Yaskawa INFORM job: FORLOOPTEST2.JBI

/JOB
//NAME FORLOOPTEST2
//POS
///NPOS 2,0,0,2,0,0
///TOOL 5
///POSTYPE PULSE
///PULSE
C00000=-3,-50477,-58433,3,-74931,486
C00001=-3,-50477,-58433,3,-74931,486
///POSTYPE ROBOT
///RECTAN
///RCONF 1,0,0,0,0,0,0,0,0,0,0,0,0,0,0,0,0,0,0,0,0,0,0,0
P00006=958.535,-37.777,-104.713,-165.2944,-7.1707,17.5149
P00007=956.377,3.321,-104.733,-165.2955,-7.1688,17.5107
//INST
///DATE 2024/03/06 15:14
///COMM For loop test
///ATTR SC,RW
///GROUP1 RB1
NOP
MOVJ C00000 VJ=3.00
FOR I001 START= 5 TO 7
	 MOVL P006 V=D[I000]
	 MOVL P007 V=5.0
NEXT I001
MOVJ C00001 VJ=3.00
END
